% RSLogix 500 project PID SUBSTITUTION LOGIC_BAK004.RSS, saved by version 8.30.00.16 %
PROJECT "UNTITLED"    % processor: Bul.1763 MicroLogix 1100 Series A %

PROGRAM FILES
  LAD 2   15 rungs

DATA FILES
  O0 OUTPUT  4 elements
  I1 INPUT  6 elements
  S2 STATUS  66 elements
  B3 BINARY  2 elements
  T4 TIMER  1 elements
  C5 COUNTER  1 elements
  R6 CONTROL  1 elements
  N7 INTEGER  5 elements
  F8 FLOAT  7 elements

LADDER 2
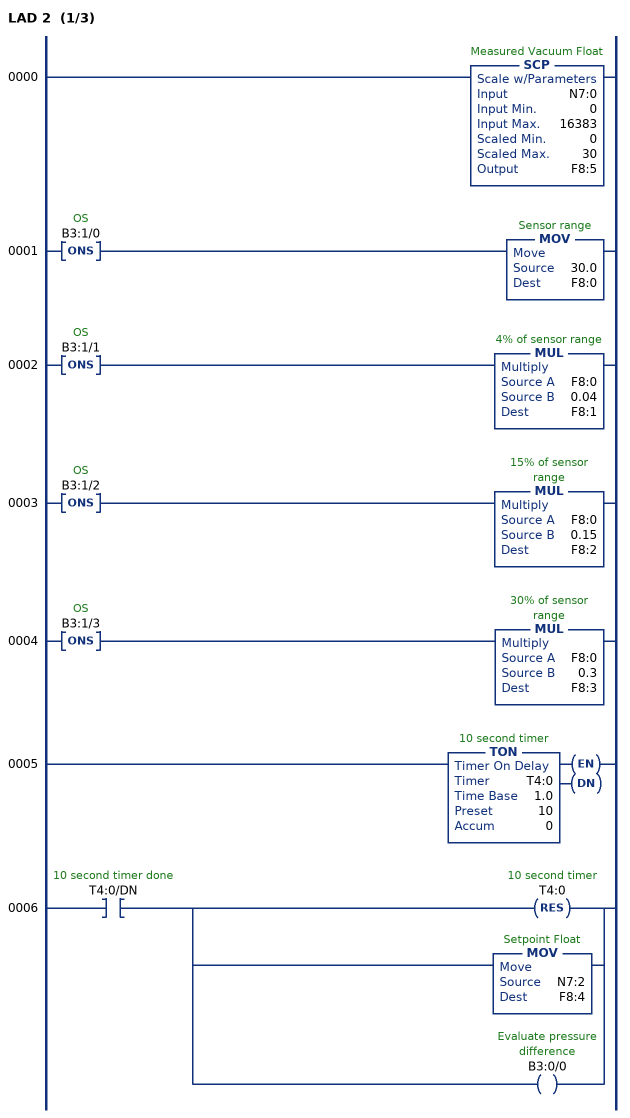
% Rung: 0 %
SOR SCP N7:0 0 16383 0 30 F8:5 EOR
%   N7:0  "Vacuum Sensor In" %
%   F8:5  "Measured Vacuum Float" %
% Rung: 1 %
SOR ONS B3:1/0 MOV 30.0 F8:0 EOR
%   B3:1/0  "OS" %
%   F8:0  "Sensor range" %
% Rung: 2 %
SOR ONS B3:1/1 MUL F8:0 0.04 F8:1 EOR
%   B3:1/1  "OS" %
%   F8:0  "Sensor range" %
%   F8:1  "4% of sensor range" %
% Rung: 3 %
SOR ONS B3:1/2 MUL F8:0 0.15 F8:2 EOR
%   B3:1/2  "OS" %
%   F8:0  "Sensor range" %
%   F8:2  "15% of sensor range" %
% Rung: 4 %
SOR ONS B3:1/3 MUL F8:0 0.3 F8:3 EOR
%   B3:1/3  "OS" %
%   F8:0  "Sensor range" %
%   F8:3  "30% of sensor range" %
% Rung: 5 %
SOR TON T4:0 1.0 10 0 EOR
%   T4:0  "10 second timer" %
% Rung: 6 %
SOR XIC T4:0/DN BST RES T4:0 NXB BST MOV N7:2 F8:4 NXB OTE B3:0/0 BND BND EOR
%   T4:0/DN  "10 second timer done" %
%   T4:0  "10 second timer" %
%   N7:2  "Vacuum Setpoint" %
%   F8:4  "Setpoint Float" %
%   B3:0/0  "Evaluate pressure difference" %

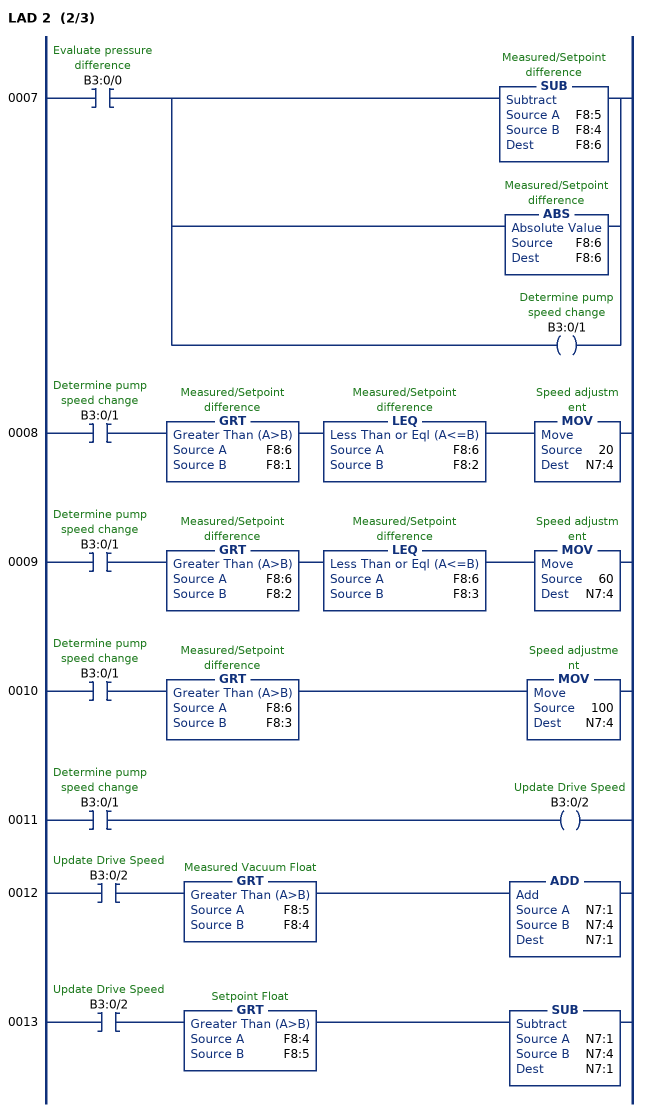
% Rung: 7 %
SOR XIC B3:0/0 BST SUB F8:5 F8:4 F8:6 NXB BST ABS F8:6 F8:6 NXB OTE B3:0/1 BND BND EOR
%   B3:0/0  "Evaluate pressure difference" %
%   F8:5  "Measured Vacuum Float" %
%   F8:4  "Setpoint Float" %
%   F8:6  "Measured/Setpoint difference" %
%   B3:0/1  "Determine pump speed change" %
% Rung: 8 %
SOR XIC B3:0/1 GRT F8:6 F8:1 LEQ F8:6 F8:2 MOV 20 N7:4 EOR
%   B3:0/1  "Determine pump speed change" %
%   F8:6  "Measured/Setpoint difference" %
%   F8:1  "4% of sensor range" %
%   F8:2  "15% of sensor range" %
%   N7:4  "Speed adjustment" %
% Rung: 9 %
SOR XIC B3:0/1 GRT F8:6 F8:2 LEQ F8:6 F8:3 MOV 60 N7:4 EOR
%   B3:0/1  "Determine pump speed change" %
%   F8:6  "Measured/Setpoint difference" %
%   F8:2  "15% of sensor range" %
%   F8:3  "30% of sensor range" %
%   N7:4  "Speed adjustment" %
% Rung: 10 %
SOR XIC B3:0/1 GRT F8:6 F8:3 MOV 100 N7:4 EOR
%   B3:0/1  "Determine pump speed change" %
%   F8:6  "Measured/Setpoint difference" %
%   F8:3  "30% of sensor range" %
%   N7:4  "Speed adjustment" %
% Rung: 11 %
SOR XIC B3:0/1 OTE B3:0/2 EOR
%   B3:0/1  "Determine pump speed change" %
%   B3:0/2  "Update Drive Speed" %
% Rung: 12 %
SOR XIC B3:0/2 GRT F8:5 F8:4 ADD N7:1 N7:4 N7:1 EOR
%   B3:0/2  "Update Drive Speed" %
%   F8:5  "Measured Vacuum Float" %
%   F8:4  "Setpoint Float" %
%   N7:4  "Speed adjustment" %
% Rung: 13 %
SOR XIC B3:0/2 GRT F8:4 F8:5 SUB N7:1 N7:4 N7:1 EOR
%   B3:0/2  "Update Drive Speed" %
%   F8:4  "Setpoint Float" %
%   F8:5  "Measured Vacuum Float" %
%   N7:4  "Speed adjustment" %

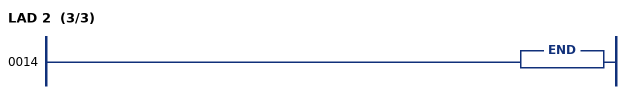
% Rung: 14 %
SOR END EOR

OTHER DOCUMENTED ADDRESSES
  B3:1/4  "OS"
  N7:3  "Measured Vacuum"
  U:3  "Control Logic"
  U:4  "Control Logic"

DATA TABLE (non-zero values as saved)
DATA T4
% .PRE .ACC %
% T4:0 % 10 0
